// Mitsubishi GX Works2 project: program_duynguyen_3phase_test   PLC: FX3U/FX3UC

PROGRAM Main
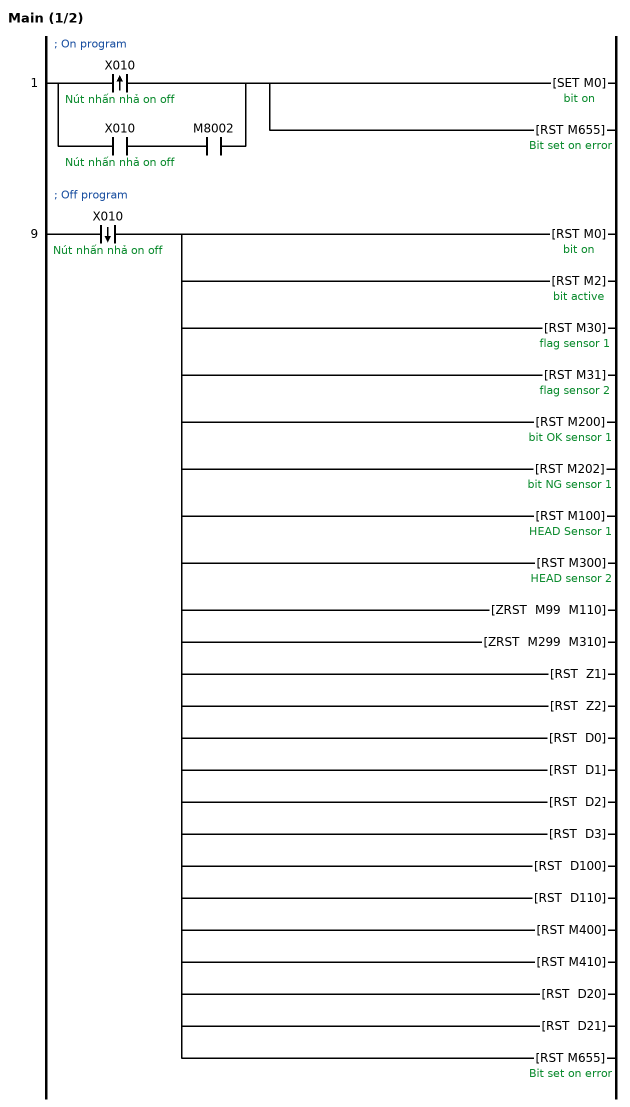
; On program
1     LDP     X010  ; Nút nhấn nhả on off
      LD      X010  ; Nút nhấn nhả on off
      AND     M8002
      ORB
      SET     M0  ; bit on
      RST     M655  ; Bit set on error
; Off program
9     LDF     X010  ; Nút nhấn nhả on off
      RST     M0  ; bit on
      RST     M2  ; bit active
      RST     M30  ; flag sensor 1
      RST     M31  ; flag sensor 2
      RST     M200  ; bit OK sensor 1
      RST     M202  ; bit NG sensor 1
      RST     M100  ; HEAD Sensor 1
      RST     M300  ; HEAD sensor 2
      ZRST    M99 M110
      ZRST    M299 M310
      RST     Z1
      RST     Z2
      RST     D0
      RST     D1
      RST     D2
      RST     D3
      RST     D100
      RST     D110
      RST     M400
      RST     M410
      RST     D20
      RST     D21
      RST     M655  ; Bit set on error
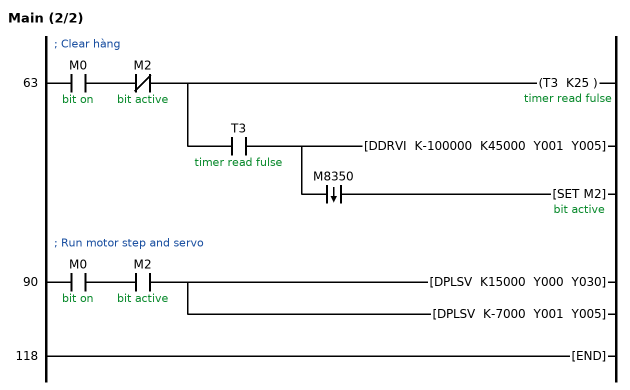
; Clear hàng
63    LD      M0  ; bit on
      ANI     M2  ; bit active
      OUT     T3 K25  ; timer read fulse
      AND     T3  ; timer read fulse
      DDRVI   K-100000 K45000 Y001 Y005
      ANDF    M8350
      SET     M2  ; bit active
; Run motor step and servo
90    LD      M0  ; bit on
      AND     M2  ; bit active
      DPLSV   K15000 Y000 Y030
      DPLSV   K-7000 Y001 Y005
118   END
END_PROGRAM

PROGRAM Trigger
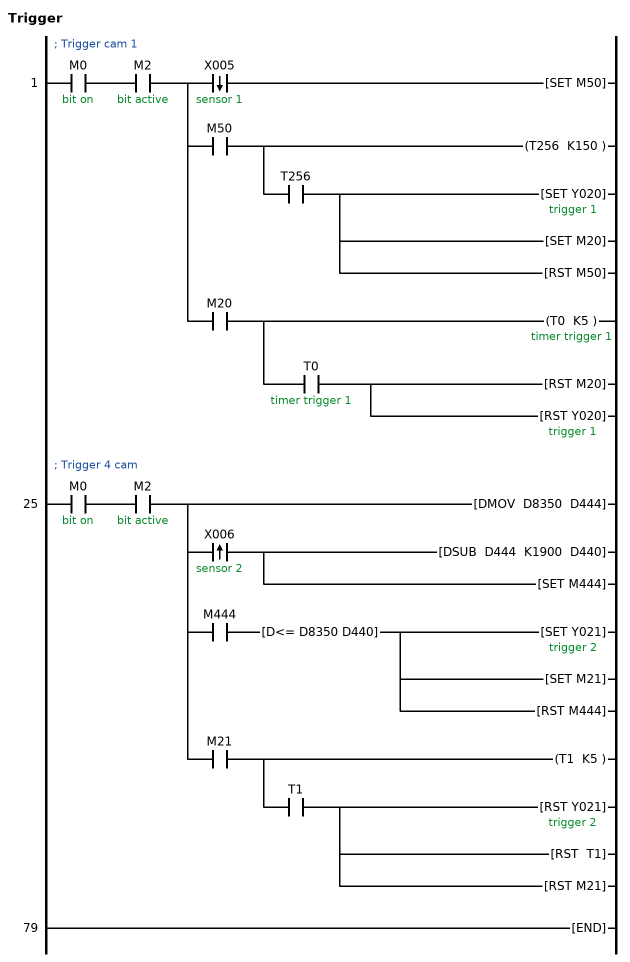
; Trigger cam 1
1     LD      M0  ; bit on
      AND     M2  ; bit active
      MPS
      ANDF    X005  ; sensor 1
      SET     M50
      MRD
      AND     M50
      OUT     T256 K150
      AND     T256
      SET     Y020  ; trigger 1
      SET     M20
      RST     M50
      MPP
      AND     M20
      OUT     T0 K5  ; timer trigger 1
      AND     T0  ; timer trigger 1
      RST     M20
      RST     Y020  ; trigger 1
; Trigger 4 cam
25    LD      M0  ; bit on
      AND     M2  ; bit active
      DMOV    D8350 D444
        [note] move ecoder to d444
      MPS
      ANDP    X006  ; sensor 2
      DSUB    D444 K1900 D440
        [note] take position after sensor 2
      SET     M444
      MRD
      AND     M444
      ANDD<=  D8350 D440
      SET     Y021  ; trigger 2
      SET     M21
      RST     M444
      MPP
      AND     M21
      OUT     T1 K5
      AND     T1
      RST     Y021  ; trigger 2
      RST     T1
      RST     M21
79    END
END_PROGRAM

PROGRAM Shiftbit
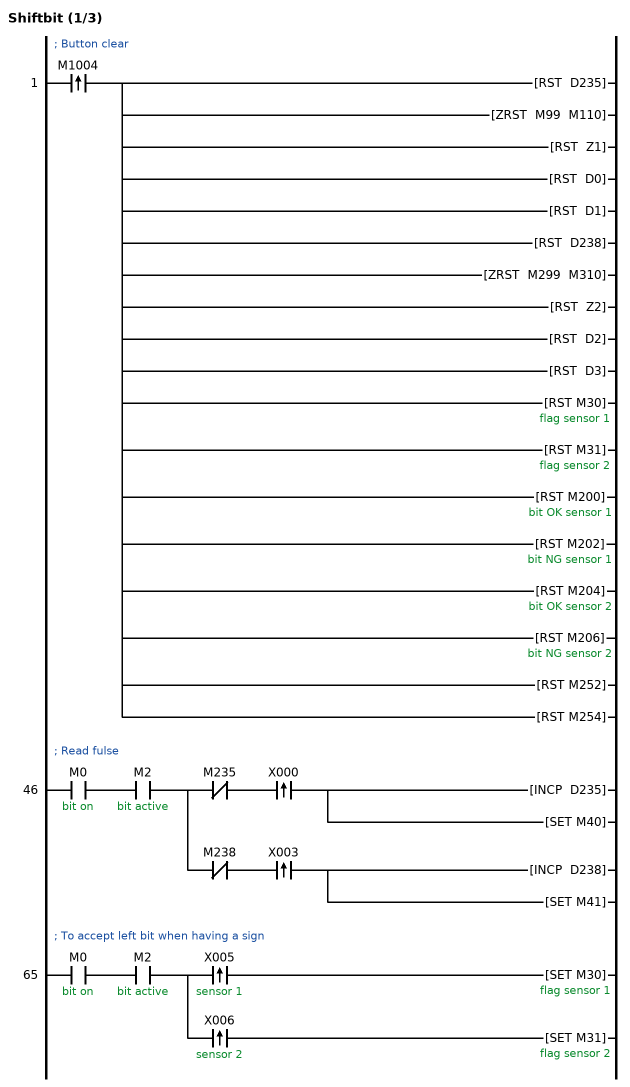
; Button clear
1     LDP     M1004
      RST     D235
      ZRST    M99 M110
      RST     Z1
      RST     D0
      RST     D1
      RST     D238
      ZRST    M299 M310
      RST     Z2
      RST     D2
      RST     D3
      RST     M30  ; flag sensor 1
      RST     M31  ; flag sensor 2
      RST     M200  ; bit OK sensor 1
      RST     M202  ; bit NG sensor 1
      RST     M204  ; bit OK sensor 2
      RST     M206  ; bit NG sensor 2
      RST     M252
      RST     M254
; Read fulse
46    LD      M0  ; bit on
      AND     M2  ; bit active
      MPS
      ANI     M235
      ANDP    X000
      INCP    D235
      SET     M40
      MPP
      ANI     M238
      ANDP    X003
      INCP    D238
      SET     M41
; To accept left bit when having a sign
65    LD      M0  ; bit on
      AND     M2  ; bit active
      MPS
      ANDP    X005  ; sensor 1
      SET     M30  ; flag sensor 1
      MPP
      ANDP    X006  ; sensor 2
      SET     M31  ; flag sensor 2
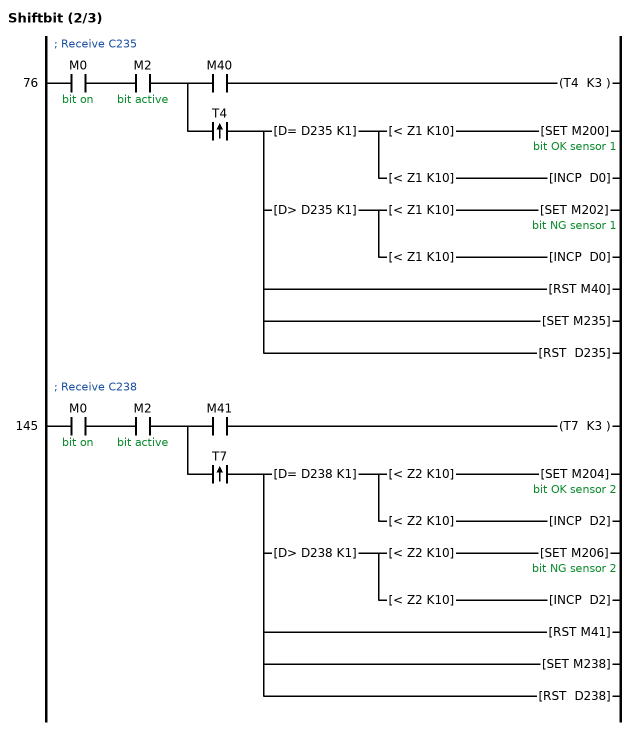
; Receive C235
76    LD      M0  ; bit on
      AND     M2  ; bit active
      MPS
      AND     M40
      OUT     T4 K3
      MPP
      ANDP    T4
      MPS
      ANDD=   D235 K1
      MPS
      AND<    Z1 K10
      SET     M200  ; bit OK sensor 1
      MPP
      AND<    Z1 K10
      INCP    D0
      MRD
      ANDD>   D235 K1
      MPS
      AND<    Z1 K10
      SET     M202  ; bit NG sensor 1
      MPP
      AND<    Z1 K10
      INCP    D0
      MPP
      RST     M40
      SET     M235
      RST     D235
; Receive C238
145   LD      M0  ; bit on
      AND     M2  ; bit active
      MPS
      AND     M41
      OUT     T7 K3
      MPP
      ANDP    T7
      MPS
      ANDD=   D238 K1
      MPS
      AND<    Z2 K10
      SET     M204  ; bit OK sensor 2
      MPP
      AND<    Z2 K10
      INCP    D2
      MRD
      ANDD>   D238 K1
      MPS
      AND<    Z2 K10
      SET     M206  ; bit NG sensor 2
      MPP
      AND<    Z2 K10
      INCP    D2
      MPP
      RST     M41
      SET     M238
      RST     D238
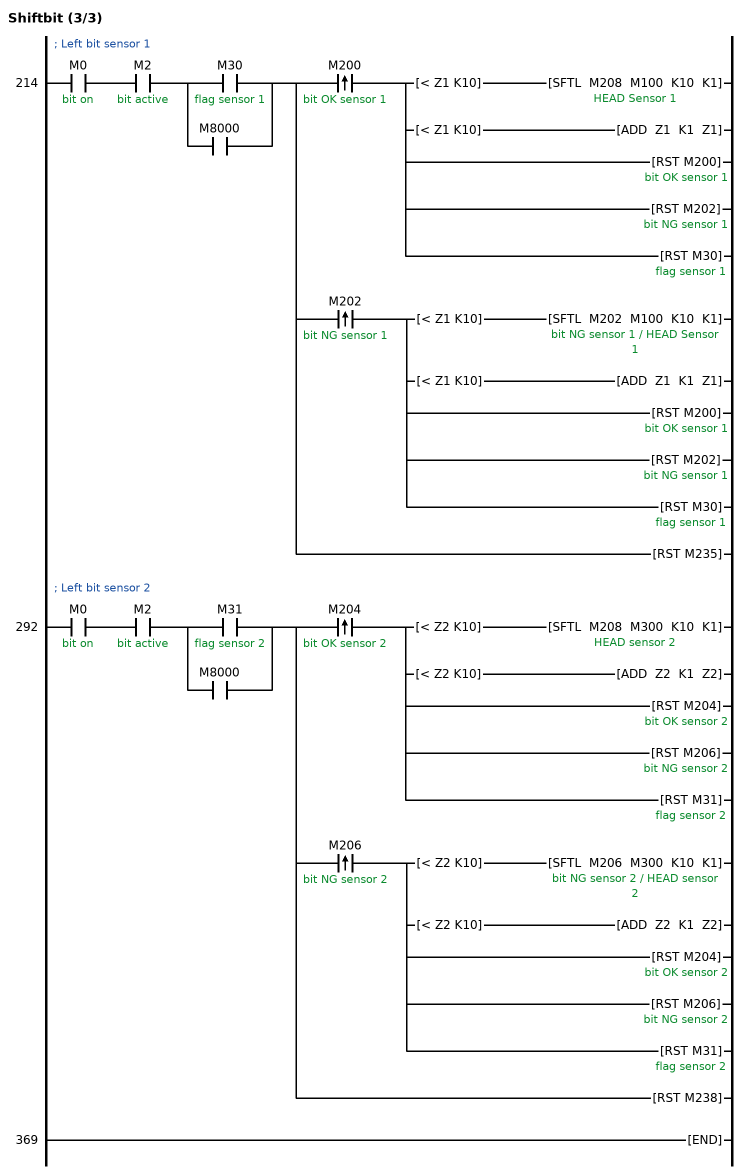
; Left bit sensor 1
214   LD      M0  ; bit on
      AND     M2  ; bit active
      LD      M30  ; flag sensor 1
      OR      M8000
      ANB
      MPS
      ANDP    M200  ; bit OK sensor 1
      MPS
      AND<    Z1 K10
      SFTL    M208 M100 K10 K1  ; HEAD Sensor 1
      MRD
      AND<    Z1 K10
      ADD     Z1 K1 Z1
      MPP
      RST     M200  ; bit OK sensor 1
      RST     M202  ; bit NG sensor 1
      RST     M30  ; flag sensor 1
      MRD
      ANDP    M202  ; bit NG sensor 1
      MPS
      AND<    Z1 K10
      SFTL    M202 M100 K10 K1
      MRD
      AND<    Z1 K10
      ADD     Z1 K1 Z1
      MPP
      RST     M200  ; bit OK sensor 1
      RST     M202  ; bit NG sensor 1
      RST     M30  ; flag sensor 1
      MPP
      RST     M235
; Left bit sensor 2
292   LD      M0  ; bit on
      AND     M2  ; bit active
      LD      M31  ; flag sensor 2
      OR      M8000
      ANB
      MPS
      ANDP    M204  ; bit OK sensor 2
      MPS
      AND<    Z2 K10
      SFTL    M208 M300 K10 K1  ; HEAD sensor 2
      MRD
      AND<    Z2 K10
      ADD     Z2 K1 Z2
      MPP
      RST     M204  ; bit OK sensor 2
      RST     M206  ; bit NG sensor 2
      RST     M31  ; flag sensor 2
      MRD
      ANDP    M206  ; bit NG sensor 2
      MPS
      AND<    Z2 K10
      SFTL    M206 M300 K10 K1
      MRD
      AND<    Z2 K10
      ADD     Z2 K1 Z2
      MPP
      RST     M204  ; bit OK sensor 2
      RST     M206  ; bit NG sensor 2
      RST     M31  ; flag sensor 2
      MPP
      RST     M238
369   END
END_PROGRAM

PROGRAM Output
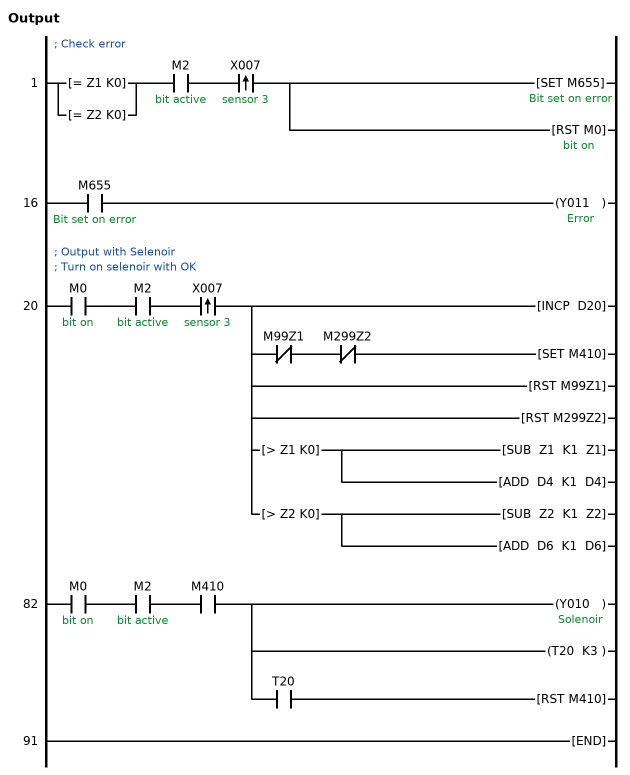
; Check error
1     LD=     Z1 K0
      OR=     Z2 K0
      AND     M2  ; bit active
      ANDP    X007  ; sensor 3
      SET     M655  ; Bit set on error
      RST     M0  ; bit on
16    LD      M655  ; Bit set on error
      OUT     Y011  ; Error
; Output with Selenoir
; Turn on selenoir with OK
20    LD      M0  ; bit on
      AND     M2  ; bit active
      ANDP    X007  ; sensor 3
      INCP    D20
      MPS
      ANI     M99Z1
      ANI     M299Z2
      SET     M410
      MPP
      RST     M99Z1
      RST     M299Z2
      MPS
      AND>    Z1 K0
      SUB     Z1 K1 Z1
      ADD     D4 K1 D4
      MPP
      AND>    Z2 K0
      SUB     Z2 K1 Z2
      ADD     D6 K1 D6
82    LD      M0  ; bit on
      AND     M2  ; bit active
      AND     M410
      OUT     Y010  ; Solenoir
      OUT     T20 K3
      AND     T20
      RST     M410
91    END
END_PROGRAM

// device comments not shown above
M1  ; bit hold
